# EPICS StreamDevice protocol: cbhv.proto
terminator = CR LF;
readtimeout = 1000;
pollperiod = 10;
replytimeout = 1000;
command {
    out "%s";
}
info {
    out "%s";
    in "%39c";
}
request {
    out "%s";
    in "%(\$1)39c";
}
spy {
    extraInput=ignore;
    in "%39c";
}
spybin {
    readtimeout = 1;
    terminator = "";
    extraInput=ignore;
    in "%r";
}
read_voltage {
    connect 1000;
    out "read_adc floats_csv %s";
    in "%20c%s";
}
set_voltage {
	    out "SetVpmF %s";
	    in "%39c";
}
